(*
SPDX-FileCopyrightText: © 2026 Oleksandr Tiutyk <trofimich@gmail.com>
SPDX-License-Identifier: MIT
License: https://opensource.org/license/mit
*)

INTERFACE IStaticCollectionFullException EXTENDS IGeneralException

METHOD Throw
VAR_INPUT
	sourceNamespaceName : STRING;
	sourceClassName : STRING;
	sourcePOUName : STRING;
	sourcePosition : STRING;
	collectionName : WSTRING;
	capacity : UDINT;
END_VAR
END_METHOD

END_INTERFACE

(* stored: Version 1.1.0.1
   Itf IStaticCollectionFullException: Id {dab6c626-d4d0-424f-8f97-94d7f340ac50}
   Method Throw: Id {1d5e094d-8546-408b-a259-af06e6c60cb7} *)
